Universal Robots PolyScope program: force_torque_tool.urp

Program force_torque_tool (createdIn=5.1.0.40195 lastSavedIn=5.1.0.40195 robotSerialNumber=2014339999 directory=/home/ur/ursim-current/programs/force torque installation=default)
Calibrated DH parameters: a=[0, -0.24355, -0.2132, 0, 0, 0]; d=[0.15185, 0, 0, 0.13105, 0.08535, 0.0921]; alpha=[1.570796, 0, 0, 1.570796, -1.570796, 0]; deltaTheta=[0, 0, 0, 0, 0, 0]
Robot Program (runOnlyOnce=true)
  force_torque := get_tcp_force()
  force_B := p[force_torque[0],force_torque[1],force_torque[2],0,0,0]
  torque_B := p[force_torque[3],force_torque[4],force_torque[5],0,0,0]
  tcp := get_actual_tcp_pose()
  rotation_BT := p[0,0,0,tcp[3],tcp[4],tcp[5]]
  force_T := pose_trans(pose_inv(rotation_BT), force_B)
  torque_T := pose_trans(pose_inv(rotation_BT), torque_B)
